FUNCTION_BLOCK SENS_VIEW (* Composite Function Block Type *)
  (* Standard: 61499-2 *)
  (* Version 0.2, 2003-12-05, JHC, Rockwell Automation, Renamed from NEWCOMPFB. *)
  (* Version 0.1, 2002-01-08, JHC, Rockwell Automation, Added DLY FB as example. *)
  (* Version 0.0, 2000-05-27, JHC, Rockwell Automation *)
  (* Compiler header: package fb.rt.vhmi; *)
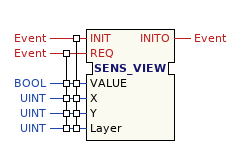
  EVENT_INPUT
    INIT WITH VALUE, X, Y, Layer; (* Initialization Request *)
    REQ WITH VALUE, X, Y, Layer; (* Normal Execution Request *)
  END_EVENT
  EVENT_OUTPUT
    INITO; (* Initialization Confirm *)
  END_EVENT
  VAR_INPUT
    VALUE : BOOL; (* Input event qualifier *)
    X : UINT;
    Y : UINT;
    Layer : UINT;
  END_VAR
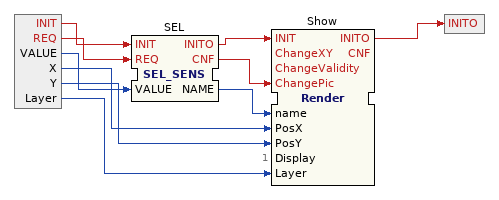
  FBS
    SEL : SEL_SENS;
    Show : Render(Display := 1);
  END_FBS
  EVENT_CONNECTIONS
    INIT TO SEL.INIT;
    REQ TO SEL.REQ;
    SEL.INITO TO Show.INIT;
    SEL.CNF TO Show.ChangePic;
    Show.INITO TO INITO;
  END_CONNECTIONS
  DATA_CONNECTIONS
    X TO Show.PosX;
    Y TO Show.PosY;
    SEL.NAME TO Show.name;
    VALUE TO SEL.VALUE;
    Layer TO Show.Layer;
  END_CONNECTIONS
END_FUNCTION_BLOCK
